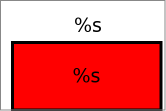
VISUALIZATION Obj_Alarm_Equipment  // 166x111
VAR_INPUT
	sIndex : STRING;
	bAlarm : BOOL;
	bOffline : BOOL;
END_VAR
    Rectangle (11,41 151x70), "%s", invisible if: bOffline
    Rectangle (10,7 156x37), "%s", text variable: sIndex
    Rectangle (11,41 151x70), "%s", colour toggle: bAlarm
END_VISUALIZATION

(* stored: Version 1.1.0.1, ProductVersion 3.1.4024.12
   Visu Obj_Alarm_Equipment: Id {0fa9a9b3-9703-4837-89af-4eea19ca38ec} *)
